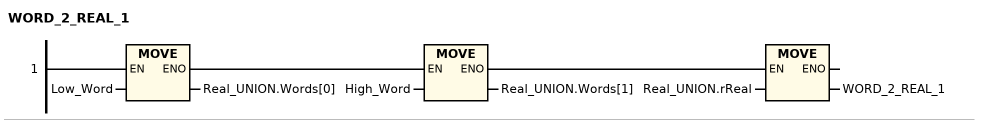
// NETWORK 1
Real_UNION.Words[0] := Low_Word;
Real_UNION.Words[1] := High_Word;
WORD_2_REAL_1 := Real_UNION.rReal;

END_FUNCTION

// 50 Functions/Word_2_Real_Div
FUNCTION Word_2_Real_Div : REAL
VAR_INPUT
	WD:WORD;
	rDIV:REAL;
END_VAR
VAR
END_VAR

// note: 1 stored wires end on pins the file does not list and are not shown
Word_2_Real_Div := WORD_TO_REAL(WD) / rDIV;

END_FUNCTION

// Library Information/GetLibVersion
// This function has been automatically generated from the project information.
FUNCTION GetLibVersion : VERSION
VAR_INPUT
	
END_VAR

GetLibVersion.uiMajor := 1;
GetLibVersion.uiMinor := 0;
GetLibVersion.uiServicePack := 0;
GetLibVersion.uiPatch := 42;

END_FUNCTION

// Library Information/GetLibVersionNumber
// This function has been automatically generated from the project information.
FUNCTION GetLibVersionNumber : DWORD
VAR_INPUT
	
END_VAR

GetLibVersionNumber := 16777258;

END_FUNCTION

// Library Information/IsLibReleased
// This function has been automatically generated from the project information.
FUNCTION IsLibReleased : BOOL
VAR_INPUT
	
END_VAR

IsLibReleased := FALSE;

END_FUNCTION

// GetBooleanProperty
// This function has been automatically generated from the project information.
{attribute 'signature_flag' := '1073741824'}
{attribute 'register_in_runtime'}
FUNCTION GetBooleanProperty : BOOL
VAR_INPUT
	stKey: WSTRING;
END_VAR

IF stKey = "IsEndUserLibrary" THEN
	GetBooleanProperty := FALSE;
ELSIF stKey = "IsStorageFormatPinned" THEN
	GetBooleanProperty := FALSE;
ELSIF stKey = "Released" THEN
	GetBooleanProperty := FALSE;
ELSE
	GetBooleanProperty := FALSE;
END_IF

END_FUNCTION

// GetCompany
// This function has been automatically generated from the project information.
{attribute 'signature_flag' := '1073741824'}
{attribute 'register_in_runtime'}
FUNCTION GetCompany : WSTRING
VAR_INPUT
	
END_VAR

GetCompany := "Burkert";

END_FUNCTION

// GetTextProperty2
// This function has been automatically generated from the project information.
{attribute 'signature_flag' := '1073741824'}
{attribute 'register_in_runtime'}
FUNCTION GetTextProperty2 : POINTER TO WSTRING
VAR_INPUT
	stKey: WSTRING;
END_VAR

IF stKey = "Author" THEN
	GetTextProperty2 := ADR("Robert Budgen");
ELSIF stKey = "Company" THEN
	GetTextProperty2 := ADR("Burkert");
ELSIF stKey = "DefaultNamespace" THEN
	GetTextProperty2 := ADR("Burkert");
ELSIF stKey = "Description" THEN
	GetTextProperty2 := ADR("");
ELSIF stKey = "LanguageModelAttribute" THEN
	GetTextProperty2 := ADR("qualified-access-only");
ELSIF stKey = "Placeholder" THEN
	GetTextProperty2 := ADR("Burkert");
ELSIF stKey = "Project" THEN
	GetTextProperty2 := ADR("Burkert");
ELSIF stKey = "Title" THEN
	GetTextProperty2 := ADR("Burkert Device Library");
ELSE
	GetTextProperty2 := ADR("");
END_IF

END_FUNCTION

// GetTextProperty
// This function has been automatically generated from the project information.
{attribute 'signature_flag' := '1073741824'}
{attribute 'register_in_runtime'}
FUNCTION GetTextProperty : WSTRING
VAR_INPUT
	stKey: WSTRING;
END_VAR

IF stKey = "Author" THEN
	GetTextProperty := "Robert Budgen";
ELSIF stKey = "Company" THEN
	GetTextProperty := "Burkert";
ELSIF stKey = "DefaultNamespace" THEN
	GetTextProperty := "Burkert";
ELSIF stKey = "Description" THEN
	GetTextProperty := "";
ELSIF stKey = "LanguageModelAttribute" THEN
	GetTextProperty := "qualified-access-only";
ELSIF stKey = "Placeholder" THEN
	GetTextProperty := "Burkert";
ELSIF stKey = "Project" THEN
	GetTextProperty := "Burkert";
ELSIF stKey = "Title" THEN
	GetTextProperty := "Burkert Device Library";
ELSE
	GetTextProperty := "";
END_IF

END_FUNCTION

// GetTitle
// This function has been automatically generated from the project information.
{attribute 'signature_flag' := '1073741824'}
{attribute 'register_in_runtime'}
FUNCTION GetTitle : WSTRING
VAR_INPUT
	
END_VAR

GetTitle := "Burkert Device Library";

END_FUNCTION

// GetVersion
// This function has been automatically generated from the project information.
{attribute 'signature_flag' := '1073741824'}
{attribute 'register_in_runtime'}
FUNCTION GetVersion : VERSION
VAR_INPUT
	
END_VAR

GetVersion.uiMajor := 1;
GetVersion.uiMinor := 0;
GetVersion.uiServicePack := 0;
GetVersion.uiPatch := 42;

END_FUNCTION

// GetVersionProperty
// This function has been automatically generated from the project information.
{attribute 'signature_flag' := '1073741824'}
{attribute 'register_in_runtime'}
FUNCTION GetVersionProperty : VERSION
VAR_INPUT
	stKey: WSTRING;
END_VAR

IF stKey = "Version" THEN
	GetVersionProperty.uiMajor := 1;
	GetVersionProperty.uiMinor := 0;
	GetVersionProperty.uiServicePack := 0;
	GetVersionProperty.uiPatch := 42;
ELSE
	GetVersionProperty.uiMajor := 0;
	GetVersionProperty.uiMinor := 0;
	GetVersionProperty.uiServicePack := 0;
	GetVersionProperty.uiPatch := 0;
END_IF

END_FUNCTION

// 20 Program Organization Units/Helpers/CalculateFrequencyWithTime
FUNCTION_BLOCK CalculateFrequencyWithTime
VAR_INPUT
    CurrentCount : DWORD;  // Current counter value
END_VAR
VAR_OUTPUT
    Frequency : REAL;      // Calculated frequency
END_VAR
VAR
    PreviousCount : DWORD; // Previous counter value
    PreviousTime : TIME;   // Previous time in milliseconds
    //CurrentTime : TIME;    // Current time in milliseconds
    PulseCount : DWORD;    // Number of pulses since the last update
    TimeDifference : REAL; // Time difference in seconds
    Timer : TON;           // Internal PLC timer for time tracking
END_VAR

// Internal PLC timer configuration (100ms base time)
Timer(IN := TRUE, PT := T#1000MS); // Trigger the timer continuously

    IF CurrentCount > PreviousCount THEN
        PulseCount := CurrentCount - PreviousCount;
        TimeDifference := TO_REAL(Timer.ET) / 1000.0;
        IF TimeDifference > 0 THEN
            Frequency := TO_REAL(PulseCount) / TimeDifference;
        ELSE
            Frequency := 0;  // Prevent division by zero
        END_IF;

        PreviousCount := CurrentCount;
		Timer(IN := FALSE);
		Timer(IN := TRUE);
	END_IF;
    
IF CurrentCount < PreviousCount THEN 
	PreviousCount:=CurrentCount; 
	Timer(IN := FALSE);
	Timer(IN := TRUE);
END_IF;

IF Timer.Q  THEN
	Frequency := 0;
	Timer(IN := FALSE);
	Timer(IN := TRUE);
END_IF;

END_FUNCTION_BLOCK

// 20 Program Organization Units/Helpers/Count_to_Hz
FUNCTION_BLOCK Count_to_Hz
VAR_INPUT
	Interval:TIME;
	Count:UDINT;
	Clear:BOOL;
END_VAR
VAR_OUTPUT
	Hz:REAL;
END_VAR
VAR
	TOF_0: TOF;
	Old_Count:UDINT;
	CLK_PULSE_0: BURKERT_OSCAT_BASIC.CLK_PULSE;
	OLD_RATE: Array[0..4] of REAL;
	
	Last_Scan: DWORD;
	History_Index:INT;
END_VAR
VAR // added by the converter: edge detectors and wires of the graphical bodies
    _w1, _w3, _w5, _w7 : BOOL;
    _w2, _w4, _w6, _w8, _w9 : UDINT;
    _w10 : ANY;
END_VAR

Last_Scan := SEL(CLK_Pulse_0.Q, Last_Scan, Burkert_OSCAT_BASIC.T_PLC_MS());
TOF_0(IN := Clear OR (Count<Old_Count), PT := T#1s); // TOF
CLK_PULSE_0(PT := Interval, N := 0, RST := TOF_0.Q); // BURKERT_OSCAT_BASIC.CLK_PULSE
_w1 := TOF_0.Q;
IF _w1 THEN _w2 := Count; END_IF
OLD_Count := _w2;
_w3 := CLK_PULSE_0.Q;
IF _w3 THEN _w4 := Count - OLD_Count; END_IF
_w5 := _w3;
IF _w5 THEN _w6 := Count; END_IF
OLD_COunt := _w6;
_w7 := _w5;
IF _w7 THEN _w8 := _w4 * (1000.0 / TIME_TO_INT(INTERVAL)); END_IF
_w9 := SEL(_w1, _w8, 0.0);
IF _w7 THEN _w10 := (History_index+1) MOD 5; END_IF
History_Index := _w10;
OLD_RATE[History_Index] := _w8;
Hz := SEL(Count<Old_Count, _w9, Hz);

END_FUNCTION_BLOCK

// 20 Program Organization Units/Helpers/FB_DilutionCalculator
FUNCTION_BLOCK FB_DilutionCalculator
VAR_INPUT
    Target_Dilution : REAL;  // Target conductivity (mS/cm, for example)
    Target_Rate : REAL; // Target flow rate (e.g., liters per second)
    Line1 : REAL;  
	Line2 :	REAL;
END_VAR

VAR_OUTPUT
    Line1_Rate : REAL; // Flow rate of the source solution
    Line2_Rate  : REAL; // Flow rate of the dilution water
    Line1_Percentage  : REAL; // Percentage of the source in the final mix
	Line2_Percentage  : REAL; // Percentage of the Water in the final mix
END_VAR

VAR
    BlendFactor:REAL;
END_VAR

IF Line1 <> Line2 THEN
    BlendFactor := (Target_Dilution - Line2) / (Line1 - Line2);

    // Ensure blend factor is within valid range (0 to 1)
    IF BlendFactor < 0 THEN
        BlendFactor := 0;
    ELSIF BlendFactor > 1 THEN
        BlendFactor := 1;
    END_IF;

    // Calculate percentages
    Line1_Percentage := BlendFactor * 100.0;
    Line2_Percentage := (1.0 - BlendFactor) * 100.0;
ELSE
    // If both conductivities are equal, split equally
    Line1_Percentage := 50.0;
    Line2_Percentage := 50.0;
END_IF;

Line1_Rate:=Target_Rate *(Line1_Percentage/100);
Line2_Rate:=Target_Rate *(Line2_Percentage/100);

END_FUNCTION_BLOCK

// 20 Program Organization Units/Helpers/FB_LookUp_Table
FUNCTION_BLOCK FB_LookUp_Table
VAR_INPUT
	VarX : REFERENCE TO ARRAY[0..19] OF REAL;
    VarY : REFERENCE TO ARRAY[0..19] OF REAL;
    ArraySize : INT;
END_VAR
VAR_OUTPUT
END_VAR
VAR
END_VAR

METHOD GetVarY : REAL
VAR_INPUT
    InputX : REAL;
END_VAR
VAR
    i : INT;
    x0, x1, y0, y1 : REAL;
END_VAR

IF ArraySize < 2 THEN
    GetVarY := 0.0;
    RETURN;
END_IF

// Extrapolate below range
IF InputX <= VarX[0] THEN
    x0 := VarX[0];
    x1 := VarX[1];
    y0 := VarY[0];
    y1 := VarY[1];
    GetVarY := y0 + ((InputX - x0) * (y1 - y0)) / (x1 - x0);
    RETURN;
END_IF

// Extrapolate above range
IF InputX >= VarX[ArraySize - 1] THEN
    x0 := VarX[ArraySize - 2];
    x1 := VarX[ArraySize - 1];
    y0 := VarY[ArraySize - 2];
    y1 := VarY[ArraySize - 1];
    GetVarY := y0 + ((InputX - x0) * (y1 - y0)) / (x1 - x0);
    RETURN;
END_IF

// Interpolate within range
FOR i := 0 TO ArraySize - 2 DO
    IF (InputX >= VarX[i]) AND (InputX <= VarX[i + 1]) THEN
        x0 := VarX[i];
        x1 := VarX[i + 1];
        y0 := VarY[i];
        y1 := VarY[i + 1];
        GetVarY := y0 + ((InputX - x0) * (y1 - y0)) / (x1 - x0);
        RETURN;
    END_IF
END_FOR
END_METHOD

END_FUNCTION_BLOCK

// 20 Program Organization Units/Helpers/FB_TempCorrection
FUNCTION_BLOCK FB_TempCorrection
VAR_INPUT
	Temp : REFERENCE TO ARRAY[0..19] OF REAL;
    Correction : REFERENCE TO ARRAY[0..19] OF REAL;
    ArraySize : INT;
END_VAR
VAR_OUTPUT
END_VAR
VAR
END_VAR

METHOD GetCorrection : REAL
VAR_INPUT
    InputTemp : REAL;
END_VAR
VAR
    i : INT;
    x0, x1, y0, y1 : REAL;
END_VAR

IF ArraySize < 2 THEN
    GetCorrection := 0.0;
    RETURN;
END_IF

// Extrapolate below range
IF InputTemp <= Temp[0] THEN
    x0 := Temp[0];
    x1 := Temp[1];
    y0 := Correction[0];
    y1 := Correction[1];
    GetCorrection := y0 + ((InputTemp - x0) * (y1 - y0)) / (x1 - x0);
    RETURN;
END_IF

// Extrapolate above range
IF InputTemp >= Temp[ArraySize - 1] THEN
    x0 := Temp[ArraySize - 2];
    x1 := Temp[ArraySize - 1];
    y0 := Correction[ArraySize - 2];
    y1 := Correction[ArraySize - 1];
    GetCorrection := y0 + ((InputTemp - x0) * (y1 - y0)) / (x1 - x0);
    RETURN;
END_IF

// Interpolate within range
FOR i := 0 TO ArraySize - 2 DO
    IF (InputTemp >= Temp[i]) AND (InputTemp <= Temp[i + 1]) THEN
        x0 := Temp[i];
        x1 := Temp[i + 1];
        y0 := Correction[i];
        y1 := Correction[i + 1];
        GetCorrection := y0 + ((InputTemp - x0) * (y1 - y0)) / (x1 - x0);
        RETURN;
    END_IF
END_FOR
END_METHOD

END_FUNCTION_BLOCK

// 20 Program Organization Units/Helpers/Flow_ETA
FUNCTION Flow_ETA : UINT
VAR_INPUT
	Target:REAL;
	Volume:REAL;
	Rate:REAL;
END_VAR
VAR
	Remain_Volume:REAL;
	Remain_minutes:REAL;
END_VAR

IF Rate >0 THEN
	Remain_Volume:=(Target-Volume);
	Remain_Minutes:=Remain_Volume/ Rate;
	Flow_Eta:=TO_UINT(Remain_Minutes*60);
ELSE
	Flow_ETA:=0;
END_IF;

END_FUNCTION

// 20 Program Organization Units/Helpers/PLC_TIME
{attribute 'hide_all_locals’}
PROGRAM PLC_TIME
VAR_INPUT
(* Change PLC Time *)
    (* User command for updating the controller's date & time *)
    i_xCmdSetDateTime           : BOOL  := FALSE;
    (* New Date: Date & Time elements for a SYSTEMDATE structure *)
    i_uiYear                    : UINT  := 2011; 
    i_uiMonth                   : UINT  :=    1; (* Mounths 1 to 12 *)
    i_uiDay                     : UINT  :=    1; (* Days 1 to 31 *)
    i_uiHour                    : UINT  :=   11; (* Hours 0 to 23 *)
    i_uiMinutes                 : UINT  :=   55; (* Minutes 0 to 59 *)
    i_uiSeconds                 : UINT  :=    0; (* Seconds 0 to 59 *)
	i_diMinuntesOffset			: DINT	:= 0; //Time Offset from UTC	
END_VAR
VAR_OUTPUT
	q_uiYear                    : UINT  := 0;
    q_uiMonth                   : UINT  := 0;
    q_uiDay                     : UINT  := 0;
    q_uiHour                    : UINT  := 0;
    q_uiMinutes                 : UINT  := 0;
    q_uiSeconds                 : UINT  := 0;
    q_uiDayOfWeek               : UINT  := 0;
    q_uiDayOfYear               : UINT  := 0;
	q_dwEpochTime				: DWORD;	
END_VAR

VAR
	(* Read PLC Time *)
    (* Result: Controller RTC as a UTC Timestamp value      *)
    (* (number of seconds since January 1st, 1970 00:00:00) *)
	{attribute 'symbol' := 'none'}
    v_dwControllerRtcAsUtc      : DWORD := 0;
    (* Result: Date & Time in a SYSTEMDATE structure *)
	{attribute 'symbol' := 'none'}
    v_PLCDate                   : SYSTIMEDATE;
    (* Result: Date & Time elements of the SYSTEMDATE structure *)
	    (* Function operation diagnostic of the "SysTimeRtcGet" function: OK if 0 *)
	{attribute 'symbol' := 'none'}
    q_udiSysTimeRtcGetDiag      : UDINT := 0;
    (* Function operation diagnostic of the "SysTimeRtcConvertUtcToDate" function: OK if 0 *)
	{attribute 'symbol' := 'none'}
    q_udiConvertUtcToDateDiag   : UDINT := 0;
(* Change PLC Time *)
    (* New Date: Date & Time as a SYSTEMDATE structure *)
	{attribute 'symbol' := 'none'}
    v_NewPLCDate                : SYSTIMEDATE;
    (* New Date: Timestamp calculated from entered Date & Time value *)
    (*  = number of seconds since January 1st, 1970 00:00:00         *)
    (*    or FFFF FFFF hex in case of unsuccessful conversion.       *)
	{attribute 'symbol' := 'none'}
    v_dwNewControllerRtcAsUtc   : DWORD := 0;
    (* Command for updating the controller's date & time: Only if they are valid *)
	{attribute 'symbol' := 'none'}
    v_xSetValidDateTime         : BOOL  := FALSE;
    (* Function operation diagnostic of the "SysTimeRtcConvertDateToUtc" function: OK if 0 *)
	{attribute 'symbol' := 'none'}
    q_udiConvertDateToUtcDiag   : UDINT := 0;
    (* Function operation diagnostic of the "SysTimeRtcSet" function: OK if 0 *)
	{attribute 'symbol' := 'none'}
    q_udiSysTimeRtcSetDiag      : UDINT := 0;
	i_diMinuntesOffset_test: DINT;
END_VAR

(*****************)
(* Read PLC Time *)
(*****************)

(* IN/OUT - Function operation diagnostic (0 if OK) *)
(* Result = Controller RTC as a UTC Timestamp value (number of seconds since January 1st, 1970 00:00:00) *)
q_dwEpochTime := SysTimeRtcGet(pResult := q_udiSysTimeRtcGetDiag);
q_dwEpochTime := DINT_TO_DWORD(DWORD_TO_DINT(q_dwEpochTime)+i_diMinuntesOffset*60);	

(* IN     - UTC Timestamp value (number of seconds since January 1st, 1970 00:00:00) *)
(* IN/OUT - Date & Time in a SYSTEMDATE structure *)
(* Result = Function operation diagnostic (OK if 0) *)
q_udiConvertUtcToDateDiag := SysTimeRtcConvertUtcToDate(dwTimestampUtc := q_dwEpochTime,  pDate:= v_PLCDate);


(* Date & Time elements of the SYSTEMDATE structure *)
(* Examples of access to any SYSTIMEDATE data: v_PLCDate => v_PLCDate.wXXXXX *)
q_uiYear        := v_PLCDate.wYear;
q_uiMonth       := v_PLCDate.wMonth;
q_uiDay         := v_PLCDate.wDay;
q_uiHour        := v_PLCDate.wHour;
q_uiMinutes     := v_PLCDate.wMinute;
q_uiSeconds     := v_PLCDate.wSecond;
q_uiDayOfWeek   := v_PLCDate.wDayOfWeek;
q_uiDayOfYear   := v_PLCDate.wYday;

(*******************)
(* Change PLC Time *)
(*******************)

(* Date & Time elements for a SYSTEMDATE structure *)
(* NOTE: The "Day of Week" and "Day of Year" elements are not useful here. *)
(* Examples of access to any SYSTIMEDATE data: v_NewPLCDate => v_NewPLCDate.wXXXXX *)
v_NewPLCDate.wYear         := i_uiYear;
v_NewPLCDate.wMonth        := i_uiMonth;
v_NewPLCDate.wDay          := i_uiDay;
v_NewPLCDate.wHour         := i_uiHour;
v_NewPLCDate.wMinute       := i_uiMinutes;
v_NewPLCDate.wSecond       := i_uiSeconds;
v_NewPLCDate.wMilliseconds := 0;

(* IN/OUT - Date & Time as a SYSTEMDATE structure *)
(* IN/OUT - New Date: Timestamp calculated from entered Date & Time value *)
(*           =  number of seconds since January 1st, 1970 00:00:00        *)
(*              or FFFF FFFF hex in case of unsuccessful conversion.      *)
(* Result = Function operation diagnostic (OK if 0) *)
q_udiConvertDateToUtcDiag := SysTimeRtcConvertDateToUtc(pDate:= v_NewPLCDate, pdwTimestampUtc := v_dwNewControllerRtcAsUtc);
v_dwNewControllerRtcAsUtc :=DINT_TO_DWORD(DWORD_TO_DINT(v_dwNewControllerRtcAsUtc)-i_diMinuntesOffset*60);

(* Command for updating the controller's date & time:            *)
(* Only if they are valid AND if in presence of the user command *)
v_xSetValidDateTime := (v_dwNewControllerRtcAsUtc <> 16#FFFFFFFF) AND i_xCmdSetDateTime;

IF v_xSetValidDateTime THEN
    (* IN     - Timestamp of the New Date (number of seconds since January 1st, 1970 00:00:00) *)
    (* Result = Function operation diagnostic (OK if 0) *)
    q_udiSysTimeRtcSetDiag := SysTimeRtcSet(ulTimestamp := v_dwNewControllerRtcAsUtc);
END_IF
i_xCmdSetDateTime:=FALSE;

END_PROGRAM

// 20 Program Organization Units/Helpers/RCP_Manager
FUNCTION RCP_Manager

VAR_IN_OUT
	Save:BOOL;
	Load:BOOL;
		Loaded:BOOL;
	Count:UINT;
END_VAR
VAR_OUTPUT

END_VAR
VAR
	RecipeManCommands:RecipeManCommands;
	Save_Response:DWORD;
	Load_Response:DWORD;
	Storage_Response:Bool;
	Load_Ton:ton;
	Save_Ton:Ton;
	Auto_Load_Ton:Ton;
	File_Save:BOOL;
	File_Save_Response:DWORD;
	//RCP_Names:ARRAY[0..9] OF STRING;
	
END_VAR
VAR
	R_Trig_0: R_Trig;
	Save_R_trig:R_trig;
END_VAR

RecipeManCommands();
Storage_Response:=RecipeManCommands.SetStoragePath('RCP/');
//RecipeManCommands.GetRecipeNames(RecipeDefinitionName:='PersistentVariables',pStrings:=ADR(RCP_Names),iSize:=10,iStartIndex:=0);
Save_R_trig(CLK:=Save);
IF Save_R_trig.Q THEN Save_Response:=16#FFFF; END_IF;


IF Save THEN 
	//Save_Response:=16#FFFF;	
	Save_Response:=ReadAndSave();
	END_IF;
IF Load THEN	Load_Response:=LoadAndWrite(); END_IF;


Save_ton(In:=Save AND NOT(Save_Response=16#FFFF),PT:=T#2S);
IF Save_Ton.Q THEN Save:=FALSE; END_IF;




Load_ton(In:=Load,PT:=T#2S);
IF Load_Ton.Q THEN		
	Load :=FALSE;
	Loaded:=TRUE;
	END_IF;

Auto_Load_Ton(IN:=NOT(Loaded),PT:=T#5S);

IF Auto_load_Ton.Q THEN Load:=TRUE;	END_IF;
//IF GVL.Day_Seconds=30500 THEN GVL.RCP_Save:=TRUE; END_IF;

R_Trig_0(CLK:=Save);
IF R_Trig_0.Q THEN	Count:=Count+1;	END_IF;



//IF File_Save THEN 
	//File_Save_Response:=RecipeManCommands.SaveRecipe	(RecipeDefinitionName:='PersistentVariables',RecipeName:='Day_27');//,FileName:='BackUp_1.txtrecipe'); 
//END_IF;

METHOD LoadAndWrite : Dword
VAR_INPUT
END_VAR
//LoadAndWrite:=RecipeManCommands.LoadAndWriteRecipe(RecipeDefinitionName:='Recipes',RecipeName:='BackUp');

LoadAndWrite:=RecipeManCommands.LoadFromAndWriteRecipe(FileName:='BackUp.Vars.txtrecipe',RecipeDefinitionName:='Vars',RecipeName:='BackUp');
END_METHOD

METHOD ReadAndSave :DWORD
VAR_INPUT
END_VAR
ReadAndSave:=RecipeManCommands.ReadAndSaveRecipe(RecipeDefinitionName:='Recipes',RecipeName:='BackUp');
//ReadAndSave:=RecipeManCommands.ReadRecipe	(RecipeDefinitionName:='PersistentVariables',RecipeName:='BackUp');


//ReadAndSave:=RecipeManCommands.ReadAndSaveRecipeAs	(RecipeDefinitionName:='PersistentVariables',RecipeName:='BackUp',FileName:='BackUp_1.txtrecipe');
END_METHOD

END_FUNCTION

// 20 Program Organization Units/Helpers/Virtual_FIT
FUNCTION_BLOCK Virtual_FIT
VAR
	Old_Total: REAL;
	OLD_V_Total: REAL;
	F_TRIG_0: F_trig;
	R_TRIG_0: R_trig;
END_VAR

VAR_OUTPUT
	V_Total:REAL;
END_VAR

VAR_INPUT
	Active:BOOL;
	Reset:BOOL;
	Total_IN:REAL;
END_VAR
VAR // added by the converter: edge detectors and wires of the graphical bodies
    _w1 : BOOL;
    _w2, _w3, _w4, _w5 : REAL;
    _w6 : ANY;
END_VAR

_w1 := Active AND (Total_In>0);
R_TRIG_0(CLK := (Total_In=0) AND Active); // R_trig
_w2 := SEL(_w1, Total_In, SEL(R_TRIG_0.Q, Old_Total, 0.0));
_w3 := SEL(_w2 >= 0.0, 0.0, _w2);
Old_Total := _w3;
_w4 := Total_In - _w3;
F_TRIG_0(CLK := Active); // F_trig
IF F_TRIG_0.Q OR Reset THEN _w5 := V_Total; END_IF
OLD_V_Total := _w5;
V_Total := _w4 + SEL(Reset, _w5, 0.0);
IF Reset THEN _w6 := 0.0; END_IF
OLD_V_Total := _w6;

END_FUNCTION_BLOCK

// 20 Program Organization Units/Level_1_Devices/FIT_Count_UDFB
FUNCTION_BLOCK FIT_Count_UDFB
VAR_INPUT
	Count:DWORD;
	//K:REAL;
	Raw_Count_16Bit:BOOL:=TRUE;
	Rate_Units:eUnits;
	Volume_Units:eUnits;
END_VAR

VAR_OUTPUT
	Reset:BOOL;
END_VAR

VAR
	R_Trig_0: R_Trig;
	COUNT_REAL: LREAL;
	Total:LREAL;
	FREQUENCY_REAL: REAL;
	Rate_Sec:REAL;
	High_Word:Word;
	ALARM_1_0: BURKERT_OSCAT_BASIC.ALARM_2;
	hihi: BOOL;
	hi: BOOL;
	lolo: BOOL;
	LO: BOOL;
	Alarm_Debounce: TON;
	//TON_0: TON;
	Pulse_500ms:Burkert_OSCAT_BASIC.CLK_PRG;
	Pulse_1s:Burkert_OSCAT_BASIC.CLK_PRG;
	tCount:DWORD;
	Analog_Alarm:Analog_Alarm_UDFB;
	Reset_Ton:TON;
	Count_Change:ARRAY[0..4] OF INT;
	Count_Index:INT;
	Ave_Hz:REAL;
	Calculate_Hz: CalculateFrequencyWithTime;
	Hz_1: REAL;
	Hz2: REAL;
	Count_2_Hz: Count_to_hz;
END_VAR
VAR_IN_OUT
	FIT:cFIT;
END_VAR

(* body of a kind this reader does not render *)

END_FUNCTION_BLOCK

// 20 Program Organization Units/Level_1_Devices/Base_Functions/Analog_Alarm_UDFB
FUNCTION_BLOCK Analog_Alarm_UDFB
VAR_INPUT
	//Config	:	REFERENCE TO cAlarm_Config;
	EU:REAL  ;
	Debounce_Active:BOOL;
	
END_VAR
VAR_OUTPUT
	Status:eSensor_Status;
	Percent_Alarm:REAL;
	
END_VAR

VAR_IN_OUT
	Config	:cAlarm_Config;
END_VAR
VAR
	Pending_Status:eSensor_Status;
	ALarm_PCT:ARRAY[0..4] OF REAL;
	//Alarm_Hold: TP;
	lclStatus:eSensor_Status;
	Alarm_Tof:TOF;
	

	
	tmp: REAL;
	Alarm_Ton:Ton;
	Warn_Ton:Ton;
END_VAR

//Status:=run();
IF Config.Mode.eMode=eHOA_Modes.Off THEN
	Status:=eSensor_Status.OK;
	Config.Within_Norms:=TRUE;
ELSE
	Eval_Alarms();

END_IF

ALarm_Tof(PT:=T#1S);


Alarm_PCT[0]:=Burkert_OSCAT_BASIC.SCALE_R(X:= EU, I_LO:= Config.Setpoints.Low_Low_Alarm - (Config.Setpoints.Low_warn-Config.Setpoints.Low_Low_Alarm), I_HI:= Config.Setpoints.Low_Low_Alarm, O_LO:=-0 , O_HI:=20 );
Alarm_PCT[1]:=Burkert_OSCAT_BASIC.SCALE_R(X:= EU, I_LO:= Config.Setpoints.Low_Low_Alarm , I_HI:= Config.Setpoints.Low_warn, O_LO:=20 , O_HI:=40 );
Alarm_PCT[2]:=Burkert_OSCAT_BASIC.SCALE_R(X:= EU, I_LO:= Config.Setpoints.Low_warn , I_HI:= Config.Setpoints.Hi_Warn, O_LO:=40 , O_HI:=60 );
Alarm_PCT[3]:=Burkert_OSCAT_BASIC.SCALE_R(X:= EU, I_LO:= Config.Setpoints.Hi_Warn , I_HI:= Config.Setpoints.Hi_Hi_Alarm, O_LO:=60 , O_HI:=80 );
Alarm_PCT[4]:=Burkert_OSCAT_BASIC.SCALE_R(X:= EU, I_LO:= Config.Setpoints.Hi_Hi_Alarm , I_HI:= Config.Setpoints.Hi_Hi_Alarm+ (Config.Setpoints.Hi_Hi_Alarm-Config.Setpoints.Hi_Warn), O_LO:=80 , O_HI:=100 );

Config.PCT_Alarm:=Alarm_PCT[2];
IF Config.Pending_Mask.0 THEN	Config.PCT_Alarm:=Alarm_PCT[0]; END_IF;
IF Config.Pending_Mask.1 THEN	Config.PCT_Alarm:=Alarm_PCT[1]; END_IF;
IF Config.Pending_Mask.5 THEN	Config.PCT_Alarm:=Alarm_PCT[3]; END_IF;
IF Config.Pending_Mask.6 THEN	Config.PCT_Alarm:=Alarm_PCT[4]; END_IF;

END_FUNCTION_BLOCK

// 20 Program Organization Units/Level_1_Devices/FIT_Rate_UDFB
FUNCTION_BLOCK FIT_Rate_UDFB
VAR_INPUT
	//Count:DWORD;
	Frequency:REAL;
	Rate_Units:eUnits;
	Volume_Units:eUnits;
END_VAR

VAR_OUTPUT
	//Reset:BOOL;
END_VAR

VAR
	Analog_Alarm:Analog_Alarm_UDFB;
	R_Trig_0: R_Trig;
	COUNT_REAL: LREAL;
	Total:LREAL;
	FREQUENCY_REAL: REAL;
	Rate_Sec:REAL;
	High_Word:Word;
	ALARM_1_0: BURKERT_OSCAT_BASIC.ALARM_2;
	hihi: BOOL;
	hi: BOOL;
	lolo: BOOL;
	LO: BOOL;
	Alarm_Debounce: TON;
	TON_0: TON;
	Pulse_1s:Burkert_OSCAT_BASIC.CLK_PRG;
	tCount:REAL;
	
END_VAR
VAR_IN_OUT
	FIT:cFIT;
	
	
END_VAR

(* body of a kind this reader does not render *)

END_FUNCTION_BLOCK

// 20 Program Organization Units/Level_1_Devices/FIT_UDFB
FUNCTION_BLOCK FIT_UDFB
VAR_INPUT
	Count:DWORD;
	Frequency:REAL;
	Raw_Count_16Bit:BOOL;
	Rate_Units:eUnits;
	Volume_Units:eUnits;
END_VAR

VAR_OUTPUT
	Reset:BOOL;
END_VAR

VAR
	Analog_Alarm:Analog_Alarm_UDFB;
	R_Trig_0: R_Trig;
	COUNT_REAL: LREAL;
	Total:LREAL;
	FREQUENCY_REAL: REAL;
	Rate_Sec:REAL;
	High_Word:Word;
	ALARM_1_0: BURKERT_OSCAT_BASIC.ALARM_2;
	hihi: BOOL;
	hi: BOOL;
	lolo: BOOL;
	LO: BOOL;
	Alarm_Debounce: TON;
	TON_0: TON;
END_VAR
VAR_IN_OUT
	FIT:cFIT;
END_VAR

(* body of a kind this reader does not render *)

END_FUNCTION_BLOCK

// 20 Program Organization Units/Level_2_Controls/Analog_Batch_Pump
FUNCTION_BLOCK Analog_Batch_Pump
VAR_INPUT
END_VAR
VAR_OUTPUT
	RUN:BOOL;
	Rev:BOOL;
	Speed:REAL;
END_VAR
VAR_IN_OUT
	Pump:cAnalog_Batch_Pump;
END_VAR
VAR
	Max_Volume:REAL;
	Min_Volume:REAL;
	TON_0: TON;
	TP_0: TP;
	TON_1: TON;
	F_TRIG_0: F_trig;
	Min_time:REAL;
	Max_Time:Real;
	New_Pump_Time: INT;
	lcl_Target:REAL;
	lcl_Seconds:REAL;
	Base_PCT: REAL;
	TON_2: TON;
	R_TRIG_0: R_trig;
	TP_1: TP;
	F_TRIG_1: F_trig;
	Cal_Value: REAL;
	RUN_REQ: BOOL;
	F_TRIG_2: F_Trig;
	TP_2: TP;
	CLK_PRG_0: BURKERT_OSCAT_BASIC.CLK_PRG;
	R_TRIG_1: R_trig;
END_VAR
VAR // added by the converter: edge detectors and wires of the graphical bodies
    _w1, _w6, _w9, _w10, _w11, _w12, _w13, _w14 : ANY;
    _w2, _w3, _w4, _w15 : REAL;
    _w5 : INT;
    _w7, _w8 : TIME;
END_VAR

Level_Manager();
_w1 := SEL(pump.Mode.eMode=eAnalog_Pump_Modes.Auto, pump.HMI_Volume_Target, pump.PLC_Volume_Target);
pump.Live_Rate := SEL(Pump.Config.Follow_ENABLE, _w1, Pump.Calibration_Rate* (pump.Config.Follow_Rate/100));
lcl_Target := _w1;
lcl_Seconds := SEL(pump.Mode.eMode=eAnalog_Pump_Modes.Auto, Pump.HMI_Volume_Target/PUMP.HMI_Rate_PCT, PUMP.PLC_Volume_Target/Pump.PLC_Rate_PCT);
_w2 := lcl_Target / ((PUMP.Config.Min_Speed/100.0) * (Pump.Calibration_Rate/60));
MAX_Time := _w2;
_w3 := lcl_Target / ((PUMP.Config.Max_Speed/100.0) * (Pump.Calibration_Rate/60));
Min_Time := _w3;
_w4 := SEL(lcl_Seconds<Min_time, SEL(lcl_Seconds>Max_Time, lcl_Seconds, _w2), _w3);
_w5 := REAL_TO_INT(_w4);
lcl_Seconds := _w5;
New_Pump_Time := _w5;
Base_PCT := SEL(lcl_Target=0, (Min_Time / _w4) * PUMP.Config.Max_Speed, 0.0);
_w6 := (Pump.Mode.eMode=eAnalog_Pump_Modes.Manual) OR Pump.PLC_Run AND (pump.Mode.eMode=eAnalog_Pump_Modes.Auto);
RUN_REQ := _w6;
_w7 := INT_TO_TIME(PUMP.Config.SuckBack_Seconds) * 1000;
_w8 := INT_TO_Time(New_Pump_Time) * 1000;
TON_0(IN := _w6, PT := _w8); // TON
_w9 := Pump.PLC_Run AND (pump.Mode.eMode=eAnalog_Pump_Modes.Auto);
_w10 := _w6 AND NOT TON_0.Q AND NOT (lcl_Target=0) OR (pump.Mode.eMode=eAnalog_Pump_Modes.Prime) OR (pump.Mode.eMode=eAnalog_Pump_Modes.Calibrate) OR Pump.Config.Follow_ENABLE;
F_TRIG_2(CLK := _w10); // F_Trig
Pump.Pump_FWD := _w10;
TP_2(IN := F_TRIG_2.Q AND (PUMP.Config.SuckBack_Seconds>1), PT := t#3s); // TP
TON_1(IN := TP_2.Q, PT := T#2s); // TON
TP_0(IN := TON_1.Q, PT := _w7); // TP
Pump.Pump_REV := TP_0.Q;
RUN := _w10 OR TP_0.Q;
REV := TP_0.Q;
PUMP.Batch_ETA := SEL(lcl_Target=0, SEL(_w6, New_Pump_time, TIME_TO_INT((_w8 - TON_0.ET) / 1000)), 0);
Pump.PCT_Remain := SEL(Run_REQ, 0.0, (1 - Pump.Volume_Delivered / pump.Live_Rate) * 100);
F_TRIG_0(CLK := _w9); // F_trig
IF F_TRIG_0.Q THEN _w11 := 0; END_IF
lcl_Target := _w11;
R_TRIG_0(CLK := Pump.Pump_FWD); // R_trig
Pump.Volume_Delivered := SEL(R_TRIG_0.Q, ((Pump.Calibration_Rate/60) * (Base_PCT/100)) * TIME_TO_INT(TON_0.ET / 1000), 0.0);
SET_Status();
F_TRIG_1(CLK := pump.Mode.eMode=eAnalog_Pump_Modes.Calibrate); // F_trig
_w12 := SEL(REV, 0, Pump.Config.SuckBack_Speed);
_w13 := (pump.HMI_Volume_Target / ((Pump.HMI_Volume_Target/ Pump.HMI_Rate_PCT) / 60.0)) * (100 / (pump.Config.Max_Speed*0.75));
Cal_Value := _w13;
IF F_TRIG_1.Q AND NOT TP_1.Q THEN _w14 := _w13; END_IF
Pump.Calibration_Rate := _w14;
_w15 := SEL(Pump.Pump_FWD, _w12, SEL(Pump.Config.Follow_ENABLE, SEL(pump.Mode.eMode=eAnalog_Pump_Modes.Prime, SEL(pump.Mode.eMode=eAnalog_Pump_Modes.Calibrate, Base_PCT, pump.Config.Max_Speed*0.75), pump.Config.Max_Speed), Pump.Config.Follow_Rate));
Pump.Pump_CV := _w15;
Speed := _w15;

END_FUNCTION_BLOCK

// 20 Program Organization Units/Level_2_Controls/Analog_Control_UDFB
FUNCTION_BLOCK Analog_Control_UDFB
VAR_INPUT
	//Raw:	REAL;

	Alarm_Enable:BOOL:=TRUE;
	Latching:BOOL:=FALSE;
	Fault:BOOL:=FALSE;
	Online:BOOL:=TRUE;
END_VAR

VAR_OUTPUT
	//Status	:BYTE;
END_VAR

VAR_IN_OUT
	Device	:Analog_Control_DUT;
END_VAR

VAR
	hihi: BOOL;
	hi: BOOL;
	lolo: BOOL;
	LO: BOOL;
	Alarm_Debounce: TON;
	deboune_Time: TIME;
	Alarm_Active: BOOL;
	Alarm_Debounce_ET: TIME;
	Alarm: BOOL;
	ALARM_2_0: BURKERT_OSCAT_BASIC.ALARM_2;
	F_TRIG_0: F_Trig;
	TON_0: TON;
END_VAR

VAR_TEMP
	EU_Range: REAL;
	Raw_Range: REAL;
	Corrected_Raw: REAL;
	Raw_Pct: REAL;
	EU_Scaled: REAL;
END_VAR
VAR // added by the converter: edge detectors and wires of the graphical bodies
    _w1 : BOOL;
END_VAR

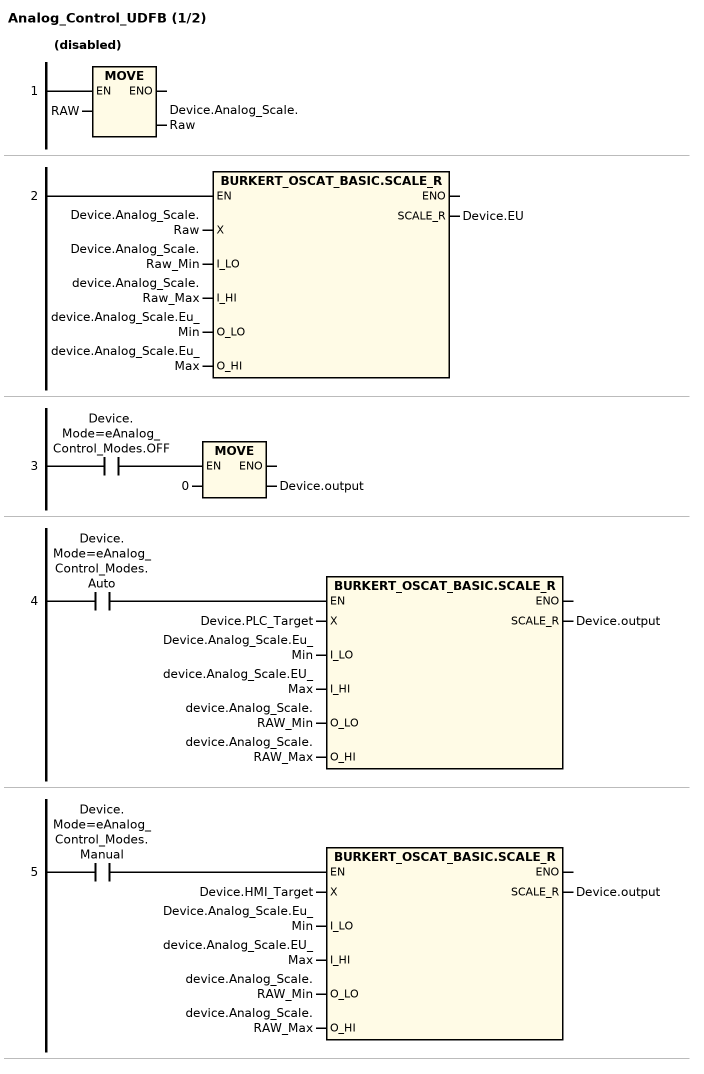
// NETWORK 1 (disabled)
// Device.Analog_Scale.Raw := RAW;

// NETWORK 2
Device.EU := BURKERT_OSCAT_BASIC.SCALE_R(X := Device.Analog_Scale.Raw, I_LO := Device.Analog_Scale.Raw_Min, I_HI := device.Analog_Scale.Raw_Max, O_LO := device.Analog_Scale.Eu_Min, O_HI := device.Analog_Scale.Eu_Max);

// NETWORK 3
IF Device.Mode=eAnalog_Control_Modes.OFF THEN Device.output := 0; END_IF

// NETWORK 4
IF Device.Mode=eAnalog_Control_Modes.Auto THEN
    Device.output := BURKERT_OSCAT_BASIC.SCALE_R(X := Device.PLC_Target, I_LO := Device.Analog_Scale.Eu_Min, I_HI := device.Analog_Scale.EU_Max, O_LO := device.Analog_Scale.RAW_Min, O_HI := device.Analog_Scale.RAW_Max);
END_IF

// NETWORK 5
IF Device.Mode=eAnalog_Control_Modes.Manual THEN
    Device.output := BURKERT_OSCAT_BASIC.SCALE_R(X := Device.HMI_Target, I_LO := Device.Analog_Scale.Eu_Min, I_HI := device.Analog_Scale.EU_Max, O_LO := device.Analog_Scale.RAW_Min, O_HI := device.Analog_Scale.RAW_Max);
END_IF

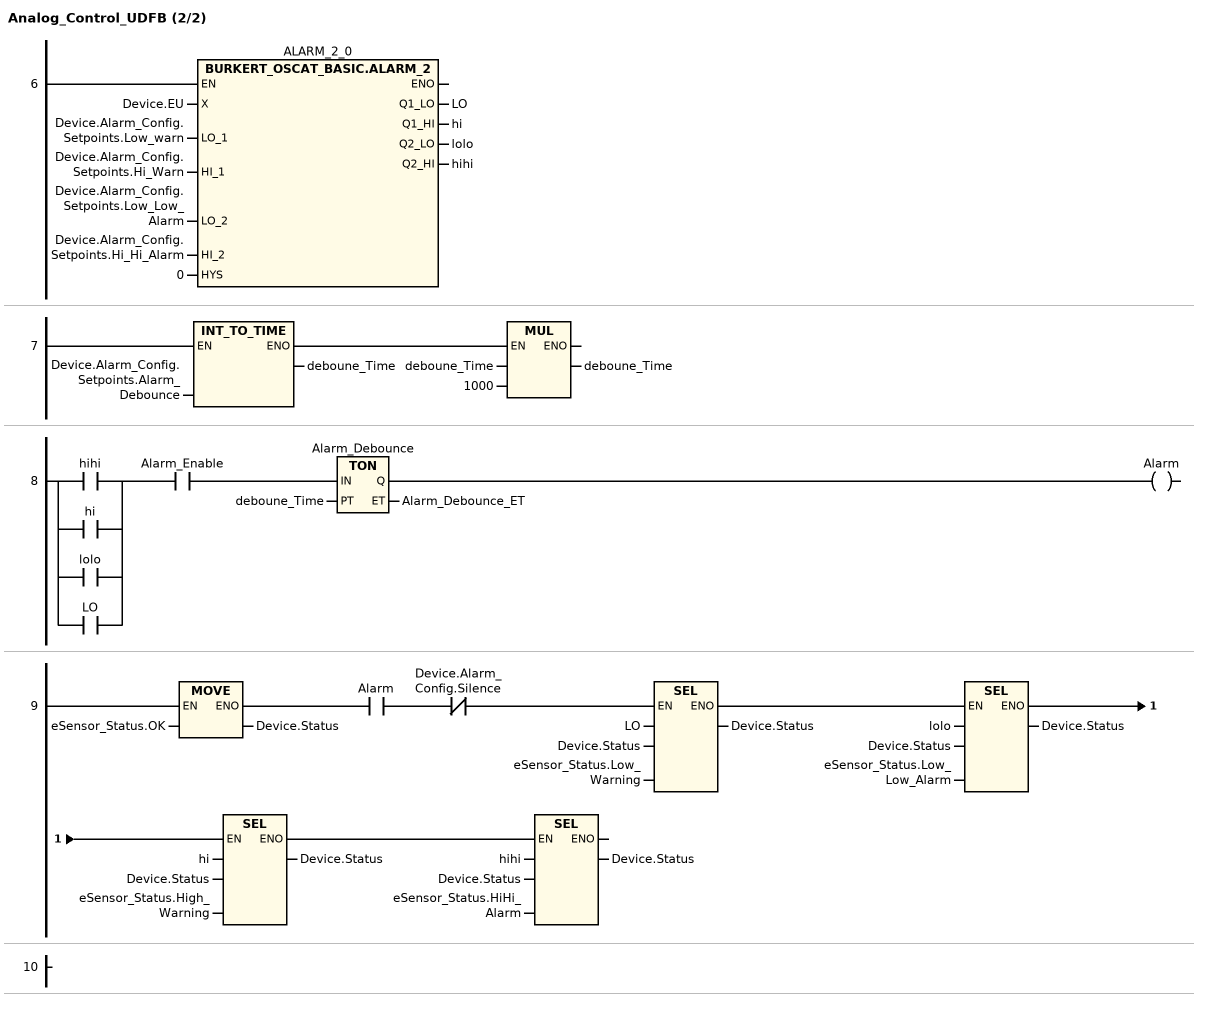
// NETWORK 6
ALARM_2_0(
    X := Device.EU,
    LO_1 := Device.Alarm_Config.Setpoints.Low_warn,
    HI_1 := Device.Alarm_Config.Setpoints.Hi_Warn,
    LO_2 := Device.Alarm_Config.Setpoints.Low_Low_Alarm,
    HI_2 := Device.Alarm_Config.Setpoints.Hi_Hi_Alarm,
    HYS := 0,
    Q1_LO => LO,
    Q1_HI => hi,
    Q2_LO => lolo,
    Q2_HI => hihi); // BURKERT_OSCAT_BASIC.ALARM_2

// NETWORK 7
deboune_Time := INT_TO_TIME(Device.Alarm_Config.Setpoints.Alarm_Debounce);
deboune_Time := deboune_Time * 1000;

// NETWORK 8
Alarm_Debounce(
    IN := (hihi OR hi OR lolo OR LO) AND Alarm_Enable,
    PT := deboune_Time,
    ET => Alarm_Debounce_ET); // TON
Alarm := Alarm_Debounce.Q;

// NETWORK 9
Device.Status := eSensor_Status.OK;
_w1 := Alarm AND NOT Device.Alarm_Config.Silence;
IF _w1 THEN Device.Status := SEL(LO, Device.Status, eSensor_Status.Low_Warning); END_IF
IF _w1 THEN Device.Status := SEL(lolo, Device.Status, eSensor_Status.Low_Low_Alarm); END_IF
IF _w1 THEN Device.Status := SEL(hi, Device.Status, eSensor_Status.High_Warning); END_IF
IF _w1 THEN Device.Status := SEL(hihi, Device.Status, eSensor_Status.HiHi_Alarm); END_IF

// NETWORK 10

END_FUNCTION_BLOCK

// 20 Program Organization Units/Level_2_Controls/Batch_Transfer
FUNCTION_BLOCK Batch_Transfer
VAR_INPUT
	//Index:INT;
	LOCK_OUT:BOOL:=FALSE;
	FIT_Rate:REAL;
	FIT_Total:REAL;
	Valve_OK:BOOL;
	Pump_OK:BOOL;	
	Destination_OK:BOOL;
END_VAR
VAR_OUTPUT
	BCV:BOOL;
	ACV:REAL;
	SFCCurrentStep:STRING;
END_VAR
VAR
	FT_PIDW_0: BURKERT_OSCAT_BASIC.FT_PIDW;
END_VAR

VAR_IN_OUT
	Transfer:cBatch_Transfer;
	FIT_Reset:BOOL;
END_VAR

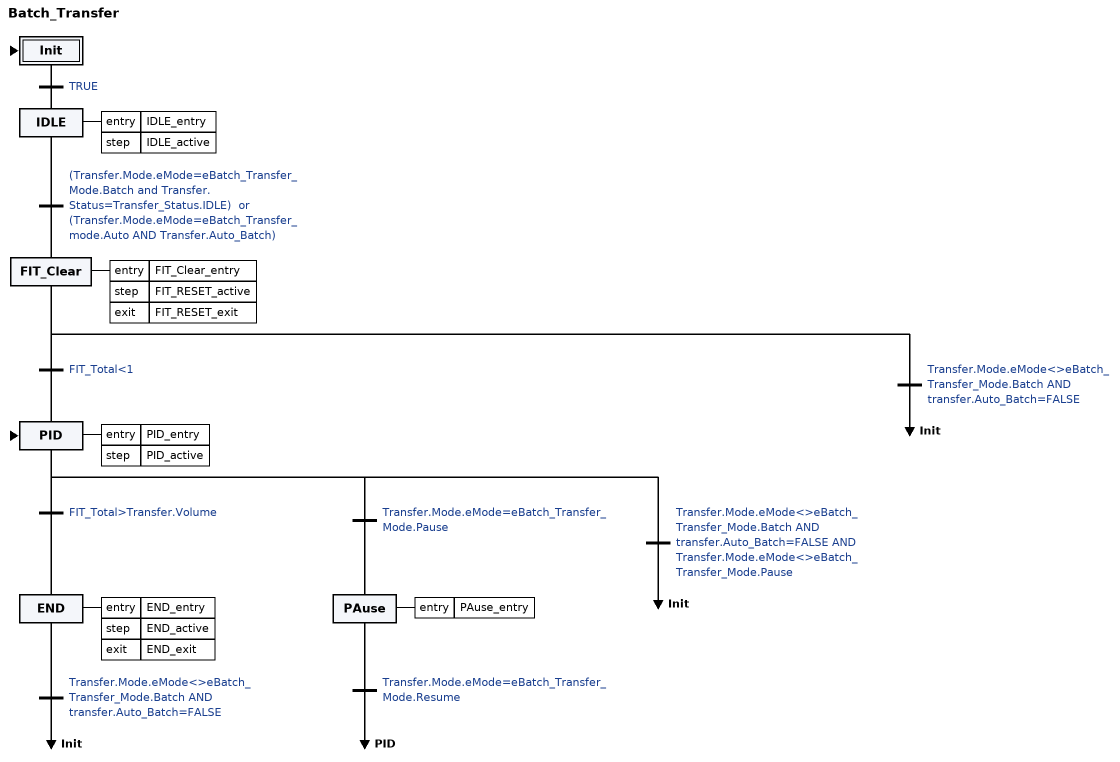
INITIAL_STEP Init:
END_STEP
TRANSITION FROM Init TO IDLE
    := TRUE;
END_TRANSITION
STEP IDLE:
    IDLE_entry(P1);  // entry action
    IDLE_active(N);  // step action
END_STEP
TRANSITION FROM IDLE TO FIT_Clear
    := (Transfer.Mode.eMode=eBatch_Transfer_Mode.Batch and Transfer.Status=Transfer_Status.IDLE) or (Transfer.Mode.eMode=eBatch_Transfer_mode.Auto AND Transfer.Auto_Batch);
END_TRANSITION
STEP FIT_Clear:
    FIT_Clear_entry(P1);  // entry action
    FIT_RESET_active(N);  // step action
    FIT_RESET_exit(P0);  // exit action
END_STEP
TRANSITION FROM FIT_Clear TO PID
    := FIT_Total<1;
END_TRANSITION
TRANSITION FROM FIT_Clear TO Init
    := Transfer.Mode.eMode<>eBatch_Transfer_Mode.Batch AND transfer.Auto_Batch=FALSE;
END_TRANSITION
STEP PID:
    PID_entry(P1);  // entry action
    PID_active(N);  // step action
END_STEP
TRANSITION FROM PID TO END
    := FIT_Total>Transfer.Volume;
END_TRANSITION
STEP END:
    END_entry(P1);  // entry action
    END_active(N);  // step action
    END_exit(P0);  // exit action
END_STEP
TRANSITION FROM END TO Init
    := Transfer.Mode.eMode<>eBatch_Transfer_Mode.Batch AND transfer.Auto_Batch=FALSE;
END_TRANSITION
TRANSITION FROM PID TO PAuse
    := Transfer.Mode.eMode=eBatch_Transfer_Mode.Pause;
END_TRANSITION
TRANSITION FROM PID TO Init
    := Transfer.Mode.eMode<>eBatch_Transfer_Mode.Batch AND transfer.Auto_Batch=FALSE AND Transfer.Mode.eMode<>eBatch_Transfer_Mode.Pause;
END_TRANSITION
STEP PAuse:
    PAuse_entry(P1);  // entry action
END_STEP
TRANSITION FROM PAuse TO PID
    := Transfer.Mode.eMode=eBatch_Transfer_Mode.Resume;
END_TRANSITION
// branch label Branch0_Run_Sequence

END_FUNCTION_BLOCK

// 20 Program Organization Units/Level_2_Controls/Chase_Master_Rate_UDFB
FUNCTION_BLOCK Chase_Master_Rate_UDFB
VAR_INPUT
	Valve_Ready:BOOL;
	Valve_Open:Bool;
END_VAR
VAR_OUTPUT
	BCV_CMD:BOOL;
	ACV_CMD:REAL;
END_VAR
VAR
	Run_Request:Bool;
	
END_VAR
VAR_IN_OUT
	chase:cChase;
	FIT:cFIT;
	Flow_PID:PID_DUT;
	//Temp_PID:PID_DUT;
END_VAR

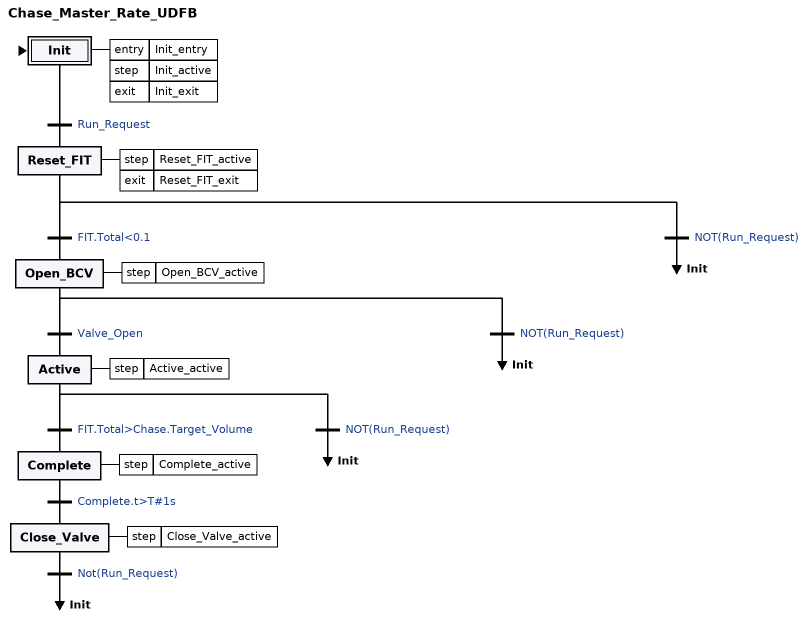
INITIAL_STEP Init:
    Init_entry(P1);  // entry action
    Init_active(N);  // step action
    Init_exit(P0);  // exit action
END_STEP
TRANSITION FROM Init TO Reset_FIT
    := Run_Request;
END_TRANSITION
STEP Reset_FIT:
    Reset_FIT_active(N);  // step action
    Reset_FIT_exit(P0);  // exit action
END_STEP
TRANSITION FROM Reset_FIT TO Open_BCV
    := FIT.Total<0.1;
END_TRANSITION
STEP Open_BCV:
    Open_BCV_active(N);  // step action
END_STEP
TRANSITION FROM Open_BCV TO Active
    := Valve_Open;
END_TRANSITION
TRANSITION FROM Open_BCV TO Init
    := NOT(Run_Request);
END_TRANSITION
STEP Active:
    Active_active(N);  // step action
END_STEP
TRANSITION FROM Active TO Complete
    := FIT.Total>Chase.Target_Volume;
END_TRANSITION
TRANSITION FROM Active TO Init
    := NOT(Run_Request);
END_TRANSITION
STEP Complete:
    Complete_active(N);  // step action
END_STEP
TRANSITION FROM Complete TO Close_Valve
    := Complete.t>T#1s;
END_TRANSITION
STEP Close_Valve:
    Close_Valve_active(N);  // step action
END_STEP
TRANSITION FROM Close_Valve TO Init
    := Not(Run_Request);
END_TRANSITION
TRANSITION FROM Reset_FIT TO Init
    := NOT(Run_Request);
END_TRANSITION

END_FUNCTION_BLOCK

// 20 Program Organization Units/Level_2_Controls/Chase_Master_UDFB
FUNCTION_BLOCK Chase_Master_UDFB
VAR_INPUT
	Valve_Ready:BOOL;
END_VAR
VAR_OUTPUT
	BCV_CMD:BOOL;
	ACV_CMD:REAL;
END_VAR
VAR
	Run_Request:Bool;
	
END_VAR
VAR_IN_OUT
	chase:cChase;
	FIT:cFIT;
	Flow_PID:PID_DUT;
	Temp_PID:PID_DUT;
END_VAR

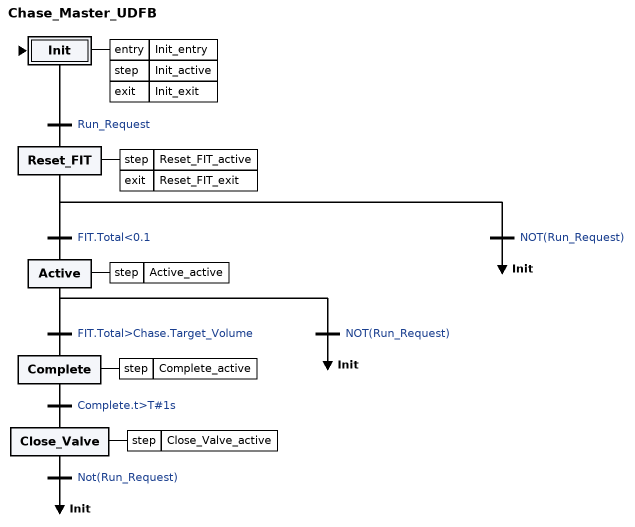
INITIAL_STEP Init:
    Init_entry(P1);  // entry action
    Init_active(N);  // step action
    Init_exit(P0);  // exit action
END_STEP
TRANSITION FROM Init TO Reset_FIT
    := Run_Request;
END_TRANSITION
STEP Reset_FIT:
    Reset_FIT_active(N);  // step action
    Reset_FIT_exit(P0);  // exit action
END_STEP
TRANSITION FROM Reset_FIT TO Active
    := FIT.Total<0.1;
END_TRANSITION
STEP Active:
    Active_active(N);  // step action
END_STEP
TRANSITION FROM Active TO Complete
    := FIT.Total>Chase.Target_Volume;
END_TRANSITION
TRANSITION FROM Active TO Init
    := NOT(Run_Request);
END_TRANSITION
STEP Complete:
    Complete_active(N);  // step action
END_STEP
TRANSITION FROM Complete TO Close_Valve
    := Complete.t>T#1s;
END_TRANSITION
STEP Close_Valve:
    Close_Valve_active(N);  // step action
END_STEP
TRANSITION FROM Close_Valve TO Init
    := Not(Run_Request);
END_TRANSITION
TRANSITION FROM Reset_FIT TO Init
    := NOT(Run_Request);
END_TRANSITION

END_FUNCTION_BLOCK

// 20 Program Organization Units/Level_2_Controls/Chase_Slave_UDFB
FUNCTION_BLOCK Chase_Slave_UDFB
VAR_INPUT
	Source_Healthy:BOOL;
	Destination_Healthy:BOOL;
	
END_VAR
VAR_OUTPUT
	BCV_CMD:BOOL;
END_VAR
VAR
	Chase_Request:BOOL;
END_VAR
VAR_IN_OUT
	Transfer:cChase;
	Chase:cChase;
END_VAR

Chase_Request:= (Chase.Mode=eChase_Mode.Auto AND Chase.PLC_Run) OR Chase.Mode=eChase_mode.Manual;
IF (Transfer.Status.eStatus=Transfer_Status.IDLE  AND Chase_Request) THEN
	Chase.Active:=TRUE;
END_IF;


IF (Transfer.Status.eStatus=Transfer_Status.IDLE AND Source_Healthy AND Destination_Healthy AND Chase_Request) OR Chase.Active THEN
	Transfer.Mode:=Chase.Mode;
	Transfer.PLC_Run:=Chase.PLC_Run;
	Transfer.Target_Rate:=Chase.Target_Rate;
	Transfer.Target_Temp:=Chase.Target_Temp;
	Transfer.Target_Volume:=Chase.Target_Volume;
	//Chase.Active:=Transfer.Active;
	Chase.Status.eStatus:=Transfer.Status.eStatus;
	Chase.PCT_Remain:=Transfer.PCT_Remain;
	Chase.ETA:=Transfer.ETA;
	BCV_CMD:=(Transfer.Status.eStatus=eChase_Status.Active);
	
ELSE
	//Chase.Active:=FALSE;
	BCV_CMD:=FALSE;
	IF NOT(Destination_Healthy) THEN
		Chase.Status.eStatus:=eChase_Status.Destination_Not_Ready;
	END_IF;
	IF NOT(Source_Healthy) THEN
		Chase.Status.eStatus:=eChase_Status.Source_Not_Ready;
	END_IF;
	IF (Transfer.Status.eStatus<>Transfer_Status.IDLE) THEN
		Chase.Status.eStatus:=eChase_Status.Not_Available;
	END_IF;
	
END_IF;

IF Chase.Active AND NOT(Chase_request) THEN
		Transfer.Mode:=Chase.Mode;
		Transfer.PLC_Run:=Chase.PLC_Run;
		Chase.Active:=FALSE;
END_IF

IF(Chase.Status.eStatus=eChase_Status.Not_Available AND Transfer.Status.eStatus=eChase_Status.IDLE) THEN
	Chase.Status.eStatus:=Transfer.Status.eStatus;
END_IF;
IF(Chase.Status.eStatus=eChase_Status.Source_Not_Ready AND Source_Healthy) THEN
	Chase.Status.eStatus:=eChase_Status.IDLE;
END_IF;
IF(Chase.Status.eStatus=eChase_Status.Destination_Not_Ready AND Destination_Healthy) THEN
	Chase.Status.eStatus:=eChase_Status.IDLE;
END_IF;

END_FUNCTION_BLOCK

// 20 Program Organization Units/Level_2_Controls/Condensate_Trap_UDFB
FUNCTION_BLOCK Condensate_Trap_UDFB
VAR_INPUT
	LSHH:BOOL;
	LSH:BOOL;
	LSL:BOOL;
	LSLL:BOOL;
	Valve_Ready:BOOL;
	
END_VAR
VAR_OUTPUT
	ACV:REAL;
END_VAR
VAR
	DI_UDFB_0: DI_UDFB;
	DI_UDFB_1: DI_UDFB;
	DI_UDFB_2: DI_UDFB;
	DI_UDFB_3: DI_UDFB;
	R_TRIG_0: R_Trig;
	Valve_Min: REAL;
	Valve_Max: REAL;
	TON_0: TON;
	TON_2: TON;
END_VAR
VAR_IN_OUT
	Trap:cCondensate_Trap;
END_VAR
VAR // added by the converter: edge detectors and wires of the graphical bodies
    _w1, _w2, _w3, _w4, _w5, _w6, _w7, _w8, _w9, _w10, _w12 : ANY;
    _w11 : BOOL;
END_VAR

DI_UDFB_1(Raw := LSH, NC_Input := False, Debounce := 500, EN_Alarm_State := True, DI := Trap.LSH); // DI_UDFB
DI_UDFB_2(Raw := LSL, NC_Input := False, Debounce := 500, EN_Alarm_State := False, DI := Trap.LSL); // DI_UDFB
_w1 := (Trap.LSL.Status.eStatus=Di_Status.Normal_Signal_Active) AND (Trap.LSLL.Status.eStatus=Di_Status.Normal_Signal_Active);
_w2 := (Trap.LSHH.Status.eStatus=Di_Status.ALARM_Signal_ACTIVE) AND (Trap.LSH.Status.eStatus=Di_Status.ALARM_Signal_ACTIVE);
DI_UDFB_3(Raw := LSLL, NC_Input := False, Debounce := 500, EN_Alarm_State := False, DI := Trap.LSLL); // DI_UDFB
IF TON_0.Q THEN _w3 := ACV+1; END_IF
_w4 := Trap.LSHH.Raw AND NOT Trap.LSH.Raw OR Trap.LSH.Raw AND NOT Trap.LSL.Raw OR Trap.LSL.Raw AND NOT Trap.LSLL.Raw;
_w5 := SEL(_w1, SEL(Trap.LSLL.Status.eStatus=Di_Status.Normal_Signal_Active, eCondensate_Status.IDLE, eCondensate_Status.Stage_1), eCondensate_Status.Stage_2);
_w6 := SEL(Trap.LSLL.Status.eStatus=Di_Status.Normal_Signal_Active, 100, Trap.Min_Valve_Positions[1]);
Trap.READY := Valve_Ready;
_w7 := SEL(_w1, _w6, Trap.Min_Valve_Positions[2]);
DI_UDFB_0(Raw := LSHH, NC_Input := False, Debounce := 500, EN_Alarm_State := True, DI := Trap.LSHH); // DI_UDFB
TON_2(IN := ACV>99, PT := T#30s); // TON
_w8 := (Trap.LSH.Status.eStatus=Di_Status.ALARM_Signal_ACTIVE) AND (Trap.LSL.Status.eStatus=Di_Status.Normal_Signal_Active);
Trap.Status := SEL(_w4, SEL(TON_2.Q, SEL(_w2, SEL(_w8, _w5, eCondensate_Status.High_Warning), eCondensate_Status.HIGH_Alarm), eCondensate_Status.Fault), eCondensate_Status.Level_Switch_Fault);
_w9 := SEL(_w2, SEL(_w8, _w7, Trap.Min_Valve_Positions[3]), 100);
_w10 := SEL(_w2, SEL(_w8, SEL(_w1, SEL(Trap.LSLL.Status.eStatus=Di_Status.Normal_Signal_Active, 0, Trap.Min_Valve_Positions[0]), Trap.Min_Valve_Positions[1]), Trap.Min_Valve_Positions[2]), Trap.Min_Valve_Positions[3]);
_w11 := _w10 <= 1;
TON_0(IN := NOT _w11 AND NOT TON_0.Q, PT := T#1s); // TON
_w12 := SEL(_w11, LIMIT(_w10, _w3, _w9), 0.0);
ACV := _w12;
TRAP.CV := _w12;

END_FUNCTION_BLOCK

// 20 Program Organization Units/Level_1_Devices/Base_Functions/DI_UDFB
FUNCTION_BLOCK DI_UDFB
VAR_INPUT
	Raw:BOOL;
	NC_Input:BOOL:=FALSE;
	Debounce:UINT:=500;
	EN_Alarm_State:BOOL:=TRUE;
END_VAR
VAR_OUTPUT
	//DI:DI_DUT;
END_VAR
VAR
	TONOF_0: BURKERT_OSCAT_BASIC.TONOF;
END_VAR
VAR_IN_OUT
	//Config:LS_Config_DUT;
END_VAR
VAR_IN_OUT
	DI:DI_DUT;
END_VAR
VAR // added by the converter: edge detectors and wires of the graphical bodies
    _w1 : TIME;
    _w2 : ANY;
    _w3 : BOOL;
END_VAR

// note: 1 stored wires end on pins the file does not list and are not shown
_w1 := UINT_TO_TIME(Debounce);
TONOF_0(IN := DI.Raw, T_ON := _w1, T_OFF := _w1); // BURKERT_OSCAT_BASIC.TONOF
_w2 := SEL(NC_INPUT AND TONOF_0.Q, SEL(NOT NC_INPUT AND NOT TONOF_0.Q, DI.Status.eStatus, DI_Status.Normal_Signal_OFF), DI_Status.Normal_Signal_Active);
DI.Raw := Raw;
_w3 := MUX(DI.Mode.eMode, TONOF_0.Q, TRUE, False);
DI.Status.eStatus := SEL(DI.MODE.eMode=DI_Modes.Forced_Off, SEL(DI.Mode.eMode=DI_Modes.Forced_On, SEL(NOT NC_Input AND TONOF_0.Q, SEL(NC_Input AND NOT TONOF_0.Q, _w2, SEL(EN_Alarm_State, Di_Status.Normal_Signal_OFF, DI_Status.Alarm_Signal_Lost)), SEL(EN_Alarm_State, Di_Status.Normal_Signal_Active, DI_Status.Alarm_Signal_Active)), DI_Status.Forced_On), DI_Status.Forced_OFF);
DI.q := _w3;

END_FUNCTION_BLOCK

// 20 Program Organization Units/Level_2_Controls/DofMaster
FUNCTION_BLOCK DofMaster
VAR_INPUT
	Config:REFERENCE TO cDOF_Master;
	ALL_Lines_Ready:BOOL;
	
END_VAR
VAR_OUTPUT
END_VAR
VAR
	R_Trig_0:R_trig;
	Batch_CLK:TON;
	R_Trig_1:R_trig;
	
END_VAR

Config.StrBatch_Mode:=Burkert_OSCAT_BASIC.REPLACE_ALL(str:=TO_STRING(Config.Batch_Mode.eMode), src:='_' , rep:=' ' );
Config.StrBatch_Status:=Burkert_OSCAT_BASIC.REPLACE_ALL(str:=TO_STRING(Config.Batch_Status.eStatus), src:='_' , rep:=' ' );
Config.StrBatch_Task:= Burkert_OSCAT_BASIC.REPLACE_ALL(str:=TO_STRING(Config.Batch_Task.eTask), src:='_' , rep:=' ' );

Config.Batch_Target_ms:=TO_UDINT((Config.Batch_Volume/Config.Batch_Rate)*60*1000);
Config.Batch_Elapsed_ms:=TO_UDINT(Batch_CLK.ET);
Config.Batch_Remain_ms:=Config.Batch_Target_ms-Config.Batch_Elapsed_ms;

R_trig_1( CLK:=(Config.Batch_Mode.eMode=eHOA_modes.Manual));

Batch_CLK(IN:=Config.Batch_Task.eTask=eBatch_Task.Run,PT:=T#6H);
Config.Batch_CLK:=Batch_CLK.ET;

IF Config.Current_Batch_Rate >0 THEN
	Config.Batch_ETA_ms:=TO_UDINT(	((Config.Batch_Volume-Config.Current_Batch_Volume) / Config.Current_Batch_Rate)*(60*1000)	);
ELSE
	Config.Batch_ETA_ms:=0;
END_IF;

IF Config.Batch_Rate >0 THEN	
	Config.Batch_Target_ms:=TO_UDINT((Config.Batch_Volume/Config.Batch_Rate)*60*1000);
	Config.Batch_Remain:=TO_TIME(		(Config.Batch_Volume/Config.Batch_Rate)*60*1000)-Config.Batch_CLK;
ELSE
	Config.Batch_Remain:=T#0MS;
	Config.Batch_Target_ms:=0;
END_IF


IF Config.Batch_Volume>0 THEN
	Config.Current_Batch_PCT:=(Config.Current_Batch_Volume/Config.Batch_Volume)*100;
ELSE
	Config.Current_Batch_PCT:=0;
	Config.Batch_Status.eStatus:=eBatch_Status.Idle;
END_IF;


IF ALL_Lines_Ready THEN
	Config.Batch_Status.eStatus:=eBatch_Status.Ready;
	IF Config.Batch_Task.eTask=eBatch_task.Resume THEN Task_resume(); END_IF;
	IF Config.Current_Batch_Rate>0.5 THEN Config.Batch_Status.eStatus:=eBatch_Status.Active; END_IF;
	
	CASE Config.Batch_Mode.eMode OF
		eHOA_Modes.Auto:
			IF Config.PLC_Run THEN 
				Config.Batch_Task.eTask:=eBatch_Task.Run; 
			ELSE
				Config.Batch_Task.eTask:=eBatch_Task.OFF;
			END_IF;
		eHOA_Modes.Manual:  
			IF R_trig_1.q	THEN	Config.Batch_Task.eTask:=eBatch_Task.Run; END_IF;
	ELSE
		Config.Batch_Task.eTask:=eBatch_Task.OFF;
		Config.Batch_Status.eStatus:=eBatch_Status.Disabled;
		Config.PLC_Run:=FALSE;
	END_CASE
ELSE
	Config.Batch_Task.eTask:=eBatch_Task.OFF;
	Config.Batch_Status.eStatus:=eBatch_Status.Fault;
	Config.Batch_Mode.eMode:=eHoa_modes.Off;
END_IF;

IF Config.Current_Batch_PCT>=100.0 OR ( Config.Current_Batch_PCT>=99.0 AND Config.Current_Batch_Rate<1) THEN Config.Batch_Status.eStatus:=eBatch_Status.Complete; END_IF;


R_Trig_0(CLK:=Config.Batch_Task.eTask=eBatch_task.Run);
IF R_Trig_0.Q THEN
	Config.MasterID:=Config.MasterID+1;
END_IF;

END_FUNCTION_BLOCK

// 20 Program Organization Units/Level_2_Controls/Duplex_VFD
FUNCTION_BLOCK Duplex_VFD
VAR_INPUT
	VFD1:REFERENCE TO VFD_CONTROL;
	VFD2:REFERENCE TO VFD_CONTROL;
	
END_VAR
VAR_OUTPUT
END_VAR
VAR
	VFD1_Primary:BOOL;
	tTime:TIME;
	Run_Ton:Ton;
	Ratio:REAL;
	Total_Run:Real;
END_VAR

VAR_IN_OUT
	Duplex:cDuplex;
END_VAR

Run_Ton(PT:=T#30D, 
	IN:= VFD1.Actual>2 OR VFD2.Actual>2);

Total_Run:=TO_REAL(Duplex.RunTime_1/1000)+TO_REAL(duplex.RunTime_2/1000);


IF (Total_Run>0) THEN	
	//Duplex.Current_Split := 50 + ((TO_REAL(Duplex.RunTime_1/1000)/TO_REAL(duplex.RunTime_2/1000))*100)/2;
	Duplex.Current_Split:=(TO_REAL(Duplex.RunTime_1/1000)/Total_Run)* 100;
END_IF;

CASE Duplex.Mode.eMode OF
	eDuplex_mode.Auto:
		IF VFD1.Actual=0 AND VFD2.Actual=0 AND Duplex.Run_Request=FALSE THEN
			VFD1_Primary:=Duplex.Current_Split<Duplex.Target_Split;
		END_IF
	eDuplex_mode.Force_1:
		VFD1_Primary:=TRUE;
	eDuplex_mode.Force_2:
		VFD1_Primary:=FALSE;
END_CASE;


IF NOT(Duplex.Run_Request) THEN
	IF VFD1_Primary THEN
		tTime:=Duplex.RunTime_1;
	ELSE
		tTime:=Duplex.RunTime_2;
	END_IF;
END_IF;



Outputs();

END_FUNCTION_BLOCK

// 20 Program Organization Units/Level_2_Controls/fb_ACV_Filter
FUNCTION_BLOCK fb_ACV_Filter
VAR_INPUT
	Config: REFERENCE TO cFilter;
	ACV_Inlet:REFERENCE TO cACV;
	ACV_Outlet:REFERENCE TO cACV;
	BCV_Vent:REFERENCE TO cBCV;
	BCV_Drain:REFERENCE TO cBCV;
	ACV_Backwash:REFERENCE TO cACV;
	//rDP:REAL;
	//Valves_OK:BOOL;
	Pressure_OK:BOOL;
	LSHH:DI_Status;
	LSLL:DI_Status;

END_VAR
VAR_OUTPUT
	

END_VAR
VAR
	Local_Status:eFilter_Status;
	Local_Mode:eFilter_Mode;
	tStatus:eFilter_Status;
	Valves_OK:BOOL;
	Auto_Prime:BOOL:=FALSE;
	Ready_Tof:TOF;
	
	
END_VAR

Config.StrMode		:=Burkert_OSCAT_BASIC.REPLACE_ALL(str:=TO_STRING(Config.Mode.eMode) , src:='_' , rep:=' ' );
Config.StrStatus 	:=Burkert_OSCAT_BASIC.REPLACE_ALL(str:=TO_STRING(Config.Status.eStatus) , src:='_' , rep:=' ' );

//DP_Alarm(Config:=Config.

Evaluate_Status();
Valves();



CASE Config.Mode.eMode OF
	eFilter_mode.Idle: Idle();
	eFilter_Mode.Prime:			Prime();
	eFilter_Mode.Active:		Active();
	eFilter_Mode.Drain:			Drain();
	eFilter_Mode.Rinse:
	eFilter_Mode.Disabled:		Disabled();
	eFilter_Mode.Maintenance:	Maintenance();
		
	
END_CASE

END_FUNCTION_BLOCK

// 20 Program Organization Units/Level_2_Controls/Filter_Pair
FUNCTION_BLOCK Filter_Pair
VAR_INPUT
	Filter: Reference to cDuplex_Filter;
END_VAR
VAR_OUTPUT
END_VAR
VAR
	Alarm:Analog_Alarm_UDFB;
	R_TRIG_0: R_trig;
	Idle_mode: R_trig;
	Filter_1_Active: R_trig;
	Filter_1_Only: R_trig;
	Filter_2_Active: R_trig;
	Filter_2_Only: R_trig;
	Filter_1x2: R_trig;
	Filter_2x1: R_trig;
	Enable_1: R_trig;
	Enable_2: R_trig;
	Non_Available: R_trig;
	Filter_1_Manual: R_trig;
	Filter_2_Manual: R_trig;
	F_Trig_1x2: F_Trig;
	F_Trig_2x1: F_Trig;
	Auto_r_trig:R_Trig;
	
	Task_ton:Ton;
	
	
	Group_Disable: R_trig;
	Group_Bypass: R_trig;
END_VAR

//Filter.DP.Alarm_Config.Silence:= (Filter.Status=eFilter_Manager_Status.Filter_1_x_2 OR Filter.Status=eFilter_Manager_Status.Filter_2_x_1);
Task_Ton(pt:=T#5S);
Alarm(Config:=Filter.DP.Alarm_Config,eu:=Filter.DP.EU,Debounce_active:=FALSE, Status=>filter.DP.Status.eStatus);


CASE Filter.Status OF
	//eFilter_Manager_Status.Idle:
	
	eFilter_Manager_Status.Enable_Filter_1:
		Task_Ton.IN:=FALSE;
		IF Filter.Filter_1.Status.eStatus=eFilter_Status.In_Service THEN  Filter.Status:=eFilter_Manager_Status.Filter_1_Active; END_IF;
		
	eFilter_Manager_Status.Filter_1_Active:
		Task_Ton.IN:=FALSE;
		IF Filter.DP.Status.eStatus=eSensor_Status.HiHi_Alarm THEN Filter.Status:=eFilter_Manager_Status.Filter_1_x_2; END_IF;
		
	eFilter_Manager_Status.Filter_1_x_2:
		Task_Ton.IN:=(Filter.Filter_1.Status.eStatus=eFilter_Status.In_Service AND Filter.Filter_2.Status.eStatus=eFilter_Status.In_Service AND NOT(Filter.DP.Status.eStatus=eSensor_Status.HiHi_Alarm));
		
		IF 	Task_Ton.Q THEN
			Filter.Status:=eFilter_Manager_Status.Filter_2_Only; 
			Filter.Filter_1.High_DP:=TRUE;
		END_IF;
	
	eFilter_Manager_Status.Enable_Filter_2:
		Task_Ton.IN:=FALSE;
		IF Filter.Filter_2.Status.eStatus=eFilter_Status.In_Service THEN  Filter.Status:=eFilter_Manager_Status.Filter_2_Active; END_IF;
	
	eFilter_Manager_Status.Filter_2_Active:
		Task_Ton.IN:=FALSE;
		IF Filter.DP.Status.eStatus=eSensor_Status.HiHi_Alarm THEN Filter.Status:=eFilter_Manager_Status.Filter_2_x_1; END_IF;
		
	eFilter_Manager_Status.Filter_2_x_1:
		Task_Ton.IN:=(Filter.Filter_1.Status.eStatus=eFilter_Status.In_Service AND Filter.Filter_2.Status.eStatus=eFilter_Status.In_Service AND NOT(Filter.DP.Status.eStatus=eSensor_Status.HiHi_Alarm) );
		IF Task_Ton.Q THEN 
			Filter.Status:=eFilter_Manager_Status.Filter_1_Only; 
			Filter.filter_2.High_DP:=TRUE;
		END_IF;
				
	eFilter_Manager_Status.Filter_1_Only:
		Task_Ton.IN:=FALSE;
		IF Filter.Filter_2.Ready AND Filter.Mode.eMode=eFilter_manager_modes.Auto THEN	
			filter.Status:=eFilter_Manager_Status.Filter_1_Active; END_IF;
	eFilter_Manager_Status.Filter_2_Only:	
		IF Filter.Filter_1.Ready AND Filter.Mode.eMode=eFilter_manager_modes.Auto THEN	
			filter.Status:=eFilter_Manager_Status.Filter_2_Active; 
		END_IF;
	
	eFilter_Manager_Status.No_Filter_Available:
		Task_Ton.IN:=FALSE;
		IF Filter.Filter_1.Ready AND Filter.Mode.eMode=eFilter_manager_modes.Auto THEN	
			filter.Status:=eFilter_Manager_Status.Filter_1_Only;
		END_IF;
		IF Filter.Filter_2.Ready AND Filter.Mode.eMode=eFilter_manager_modes.Auto THEN	
			filter.Status:=eFilter_Manager_Status.Filter_2_Only;
		END_IF;
		
	eFilter_Manager_Status.Disabled:
		Filter.Filter_1.Status.eStatus:=eFilter_Status.Disabled;
		Filter.Filter_2.Status.eStatus:=eFilter_Status.Disabled;
		//eFilter_Manager_Status.No_Filter_Available:
	
END_CASE

Mode();
Filter_Control();



filter.strStatus:=Burkert_OSCAT_BASIC.REPLACE_ALL(str:=TO_STRING(Filter.Status), src:='_' , rep:=' ' );

END_FUNCTION_BLOCK

// 20 Program Organization Units/Level_2_Controls/HighSpeed_Tempered
FUNCTION_BLOCK HighSpeed_Tempered
VAR_INPUT
	Line: REFERENCE TO HighSpeed_Tempered_Line;
	
	CW1:REFERENCE TO ACV_DUT;
	CW2:REFERENCE TO ACV_DUT;
	HW1:REFERENCE TO ACV_DUT;
	HW2:REFERENCE TO ACV_DUT;
	
	CW_Inlet_Pressure:REAL;
	CW_Outlet_Pressure:REAL;
	
	HW_Inlet_Pressure:REAL;
	HW_Outlet_Pressure:REAL;
	HW_Supply_Temp:REAL;
	HW_Outlet_Temp:REAL;
	CW_Supply_Temp:REAL;
	CW_Outlet_Temp:REAL;
	HW_Flow:REAL;
	CW_Flow:REAL;
	Combined_Temp:REAL;
	Combined_Flow:REAL;
	
	
END_VAR
VAR_OUTPUT
	
END_VAR
VAR
	Local_Task:eHighspeed_Tempered_Task;
	Local_Status:eHighSpeed_Tempered_Status;
	Task_Ton:TON;
	
	FlowIndex, TempIndex : INT;
	
	CW_SH_1:Burkert_OSCAT_BASIC.SH_1;
	HW_SH_1:Burkert_OSCAT_BASIC.SH_1;
	CW_AVG:Burkert_OSCAT_BASIC.FT_AVG;
	HW_AVG:Burkert_OSCAT_BASIC.FT_AVG;
	
	
END_VAR

Math();
Task_Ton();

IF Line.Mode.eMode=eHighSpeed_Tempered_mode.OFF THEN
	Line.Task.eTask:=eHighSpeed_Tempered_Task.OFF;
END_IF;

CASE Line.Task.eTask OF
	
	eHighSpeed_Tempered_Task.OFF:Task_OFF();
	eHighSpeed_Tempered_Task.Calibrate:
		//Task_Calibrate();
	eHighSpeed_Tempered_Task.Run:
	
	
END_CASE

END_FUNCTION_BLOCK

// 20 Program Organization Units/Level_2_Controls/MixLine_PCT
FUNCTION_BLOCK MixLine_PCT EXTENDS Batch
VAR_INPUT
	Master:REFERENCE TO cDOF_Master;
	MixLine:REFERENCE TO cDOF_Line_PCT;
	
	
END_VAR
VAR_OUTPUT
END_VAR
VAR
	PCT_Error:REAL;
	Rate_Gain:REAL;

END_VAR

Config REF=MixLine;
Config.Batch_Volume:=	Master.Batch_Volume *(MixLine.Target_PCT/100);
Config.Batch_Rate := 	Master.Batch_Rate * (MixLine.Target_PCT/100);
MixLine.Live_Target_Volume:=(Config.Batch_Volume *(Master.Current_Batch_PCT/100));



PCT_Error:=(MixLine.Target_PCT- MixLine.Live_PCT);
Rate_Gain := 1+(PCT_Error*MixLine.Rate_KP);

MixLine.PLC_Run:=Master.PLC_Run;


CASE Master.Batch_Task.eTask OF
	eBatch_Task.Run:
		Config.Line_Task.eTask:=eBatch_Task.Run;
		IF Config.Line_Status.eStatus=eBatch_Status.Paused THEN Local_Status:=eBatch_Status.Active; END_IF;
		
		CASE Config.Line_Status.eStatus OF
			eBatch_Status.Starting:
				//Task_Run();
			eBatch_status.Active:
				Config.Batch_Rate:=	LIMIT (Config.Min_Rate,	(Config.Batch_Rate	*Rate_Gain), Config.Max_Rate);
				//Task_Run();
		END_CASE
		IF Master.Current_Batch_Volume >= MixLine.Start_Point THEN
			MixLine.Live_PCT:=((Config.Actual_Volume/Master.Current_Batch_Volume)*100);
			Task_Run();
		END_IF;
	eBatch_task.Pause:
		Task_Pause();
	eBatch_Task.Resume:
		Task_resume();
		
	eBatch_task.OFF:
		Task_OFF();
		MixLine.Live_PCT:=0;
		Config.Line_Task.eTask:=eBatch_Task.OFF;
		
ELSE
	Task_OFF();
	Config.Line_Task.eTask:=eBatch_Task.OFF;
	MixLine.Live_PCT:=0;
END_CASE

IF NOT(MixLine.Live_PCT=MixLine.Live_PCT) THEN MixLine.Live_PCT:=0; END_IF;

END_FUNCTION_BLOCK

// 20 Program Organization Units/Level_2_Controls/MixLine_Time
FUNCTION_BLOCK MixLine_Time EXTENDS Batch
VAR_INPUT
	Master:REFERENCE TO cDOF_Master;
	MixLine:REFERENCE TO cDOF_Line_PCT;
	
END_VAR
VAR_OUTPUT
END_VAR
VAR
	Rate_Error:REAL;
	Rate_Gain:REAL;
	Ramp_0:RAMP_REAL;
END_VAR

Config REF=MixLine;
Config.Batch_Volume:=	Master.Batch_Volume *(MixLine.Target_PCT/100);
Config.Batch_Rate := 	Master.Batch_Rate * (MixLine.Target_PCT/100);
MixLine.Live_Target_Volume:=(Config.Batch_Volume *(Master.Current_Batch_PCT/100));



Rate_Error:=(MixLine.Target_PCT- MixLine.Live_PCT);
Rate_Gain := 1+(Rate_Error*MixLine.Rate_KP);

MixLine.PLC_Run:=Master.PLC_Run;


CASE Master.Batch_Task.eTask OF
	eBatch_Task.Run:
		
		Config.Line_Task.eTask:=eBatch_Task.Run;
		IF Config.Line_Status.eStatus=eBatch_status.Active THEN
			Ramp_0.IN:=	LIMIT (Config.Min_Rate,	(Config.Batch_Rate	*Rate_Gain), Config.Max_Rate);
			Config.Batch_Rate:=	LIMIT (Config.Min_Rate,	(Config.Batch_Rate	*Rate_Gain), Config.Max_Rate);
		END_IF;
		IF Master.Current_Batch_Volume >= MixLine.Start_Point THEN
			MixLine.Live_PCT:=((Config.Actual_Volume/Master.Current_Batch_Volume)*100);
			Task_Run();
		END_IF;
ELSE
	Task_OFF();
	Config.Line_Task.eTask:=eBatch_Task.OFF;
	MixLine.Live_PCT:=0;
	Ramp_0.IN:=Config.Batch_Rate;
END_CASE

END_FUNCTION_BLOCK

// 20 Program Organization Units/Level_2_Controls/PID_UDFB
FUNCTION_BLOCK PID_UDFB
VAR_INPUT
	Reverse:BOOL;
	CV_OK:BOOL;
	PV_OK:BOOL;
END_VAR
VAR_OUTPUT
	CV:REAL;
END_VAR
VAR
	FT_PIDW_0: BURKERT_OSCAT_BASIC.FT_PIDW;
	R_TRIG_0: R_trig;
	Loop_Enable: BOOL;
	R_TRIG_1: R_Trig;
END_VAR
VAR_IN_OUT
	PID:PID_DUT;
END_VAR
VAR // added by the converter: edge detectors and wires of the graphical bodies
    _w1, _w2, _w3, _w4, _w6, _w7 : ANY;
    _w5 : BOOL;
END_VAR

